// TIA Portal V21 program export: 0 tag tables, 1 data types, 3 data blocks, 10 code blocks (in call order from the OBs), 0 instance data blocks

TYPE "Dane"
   STRUCT
      z1 : Bool;
      z2 : Bool;
      "string" : String;
   END_STRUCT;
END_TYPE

DATA_BLOCK "12312"   // DB2
{ S7_Optimized_Access := 'TRUE' }
   VAR
      wad : Real;
      xawd : Bool;
   END_VAR
BEGIN
END_DATA_BLOCK

DATA_BLOCK "Data_block_1"   // DB1
{ S7_Optimized_Access := 'TRUE' }
   VAR
      "zmienna 1" : Bool;
      "zmienna 2" : Bool;
   END_VAR
BEGIN
END_DATA_BLOCK

DATA_BLOCK "Dzieleniedb"   // DB3
{ S7_Optimized_Access := 'TRUE' }
   VAR
      z1 : Real;
      z2 : Real := 30.0;
      wynik : Real;
   END_VAR
BEGIN
END_DATA_BLOCK

ORGANIZATION_BLOCK "Main"   // OB1, LAD, ProgramCycle
TITLE = "Main Program Sweep (Cycle)"
{ S7_Optimized_Access := 'TRUE' }
// stored: SetENOAutomatically false
BEGIN

REGION Network 2 (SCL)
   "Data_block_1"."zmienna 1" := "Data_block_1"."zmienna 2";
END_REGION
END_ORGANIZATION_BLOCK

FUNCTION "Block_1wadawd" : Void   // FC1, LAD
{ S7_Optimized_Access := 'TRUE' }
// stored: SetENOAutomatically false
BEGIN
END_FUNCTION

FUNCTION "Dodawanie" : Void   // FC2, LAD
{ S7_Optimized_Access := 'TRUE' }
// stored: SetENOAutomatically false
BEGIN

REGION Network 1
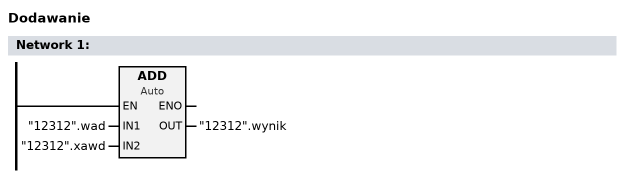
   RUNG wire#powerrail
      { S7_GenerateENO := "TRUE" } Add(in1 := "12312".wad, in2 := "12312".xawd, out => "12312".wynik)
   END_RUNG
   // the same network as SCL:
   "12312".wynik := "12312".wad + "12312".xawd;
END_REGION
END_FUNCTION

FUNCTION "Dzielenie" : Void   // FC3, LAD
{ S7_Optimized_Access := 'TRUE' }
// stored: SetENOAutomatically false
BEGIN

REGION Network 1
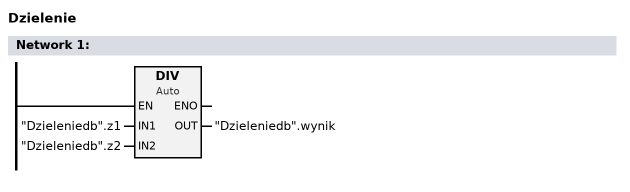
   RUNG wire#powerrail
      { S7_GenerateENO := "TRUE" } Div(in1 := "Dzieleniedb".z1, in2 := "Dzieleniedb".z2, out => "Dzieleniedb".wynik)
   END_RUNG
   // the same network as SCL:
   "Dzieleniedb".wynik := "Dzieleniedb".z1 / "Dzieleniedb".z2;
END_REGION
END_FUNCTION

FUNCTION "Nowy_blok" : Void   // FC1, LAD
{ S7_Optimized_Access := 'TRUE' }
// stored: SetENOAutomatically false
BEGIN
END_FUNCTION

FUNCTION "Odejmowanie" : Void   // FC4, LAD
{ S7_Optimized_Access := 'TRUE' }
// stored: SetENOAutomatically false
BEGIN
END_FUNCTION

FUNCTION "chuj" : Void   // FC8, LAD
{ S7_Optimized_Access := 'TRUE' }
// stored: SetENOAutomatically false
BEGIN

REGION Network 1
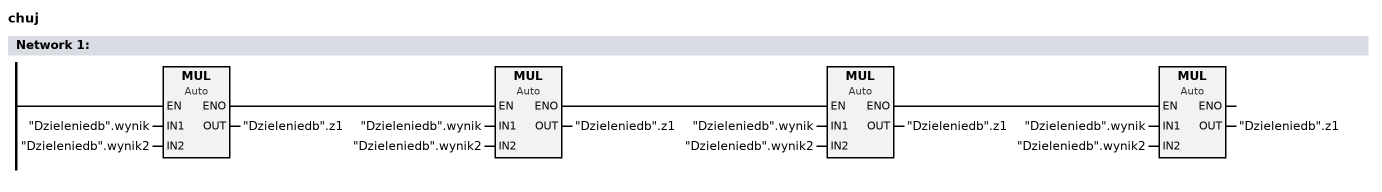
   RUNG wire#powerrail
      { S7_GenerateENO := "TRUE" } Mul(in1 := "Dzieleniedb".wynik, in2 := "Dzieleniedb".wynik2, out => "Dzieleniedb".z1)
      { S7_GenerateENO := "TRUE" } Mul(in1 := "Dzieleniedb".wynik, in2 := "Dzieleniedb".wynik2, out => "Dzieleniedb".z1)
      { S7_GenerateENO := "TRUE" } Mul(in1 := "Dzieleniedb".wynik, in2 := "Dzieleniedb".wynik2, out => "Dzieleniedb".z1)
      { S7_GenerateENO := "TRUE" } Mul(in1 := "Dzieleniedb".wynik, in2 := "Dzieleniedb".wynik2, out => "Dzieleniedb".z1)
   END_RUNG
   // the same network as SCL:
   // ENO of a box is taken as its EN; it also drops when the box reports an error
   "Dzieleniedb".z1 := "Dzieleniedb".wynik * "Dzieleniedb".wynik2;
   "Dzieleniedb".z1 := "Dzieleniedb".wynik * "Dzieleniedb".wynik2;
   "Dzieleniedb".z1 := "Dzieleniedb".wynik * "Dzieleniedb".wynik2;
   "Dzieleniedb".z1 := "Dzieleniedb".wynik * "Dzieleniedb".wynik2;
END_REGION
END_FUNCTION

FUNCTION "gbbbbbb" : Void   // FC5, LAD
{ S7_Optimized_Access := 'TRUE' }
// stored: SetENOAutomatically false
BEGIN
END_FUNCTION

FUNCTION "vawdawdwad" : Void   // FC7, LAD
{ S7_Optimized_Access := 'TRUE' }
// stored: SetENOAutomatically false
BEGIN
END_FUNCTION

FUNCTION "xwaxwadfawd" : Void   // FC6, LAD
{ S7_Optimized_Access := 'TRUE' }
// stored: SetENOAutomatically false
BEGIN
END_FUNCTION
